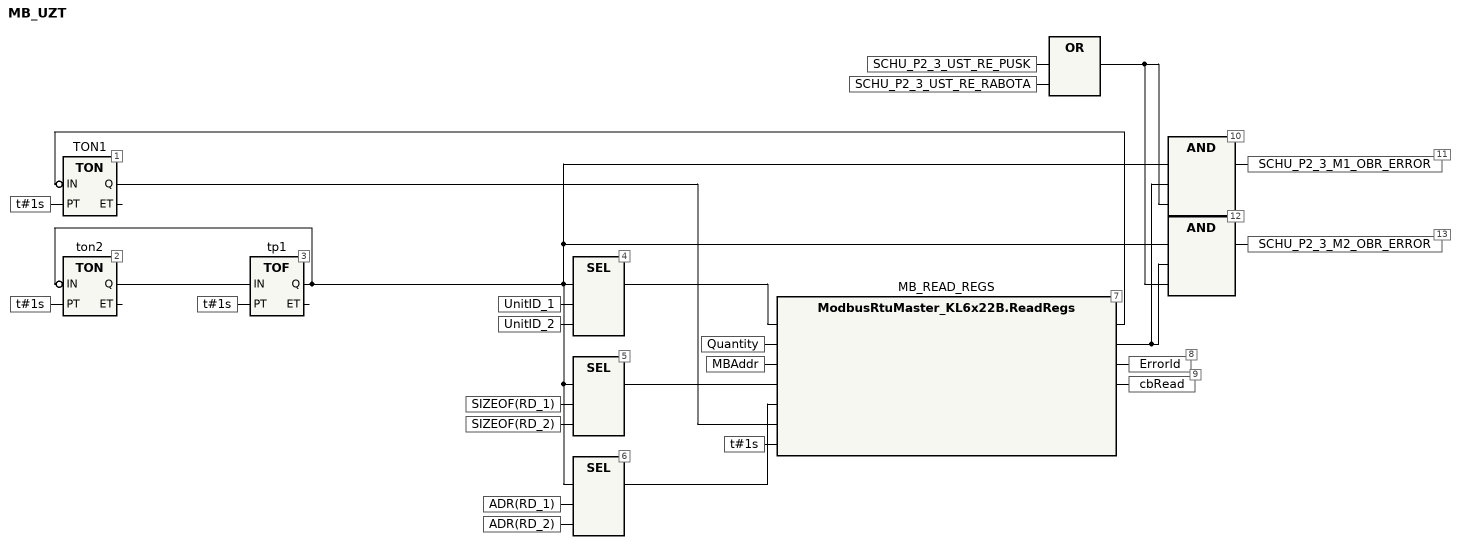
[picture p552: MB_UZT (CFC)]
_CFC_ (* Continuous Function Chart, elements in execution order *)
#0 OR(SCHU_P2_3_UST_RE_PUSK, SCHU_P2_3_UST_RE_RABOTA)
#1 TON1:TON(IN: NOT #7.out 1, PT: t#1s)
#2 ton2:TON(IN: NOT #3.Q, PT: t#1s)
#3 tp1:TOF(IN: #2.Q, PT: t#1s)
#4 SEL(#3.Q, UnitID_1, UnitID_2)
#5 SEL(#3.Q, SIZEOF(RD_1), SIZEOF(RD_2))
#6 SEL(#3.Q, ADR(RD_1), ADR(RD_2))
#7 MB_READ_REGS:ModbusRtuMaster_KL6x22B.ReadRegs(#4, Quantity, MBAddr, #5, #6, #1.Q, t#1s)
#8 Errorld <= #7.out 3
#9 cbRead <= #7.out 4
#10 AND(#3.Q, #7.out 2, #0)
#11 SCHU_P2_3_M1_OBR_ERROR <= #10
#12 AND(#3.Q, #7.out 2, #0)
#13 SCHU_P2_3_M2_OBR_ERROR <= #12
_END_CFC_
END_PROGRAM

(* POU IM/YA1_Upr_1, CFC *)
PROGRAM YA1_Upr_1
VAR
	RS_YA1_Open: RS;
	RT_Pusk: R_TRIG;
	RT_OSTANOV: R_TRIG;
	fb_HVACPA: FB_HVAC2PointActuator;

	stokeTime: TIME;
	enableLimitSwitch: BOOL := TRUE;
	FT_PCH_OTKL: R_TRIG;
	TON_PCH_OTKL: TON;
	ZADERJ_SHOD_YA1: TON;
	TON_YA1_Z_ZAM_TE2: TON;
	TON_OTK_MV: TON;
END_VAR
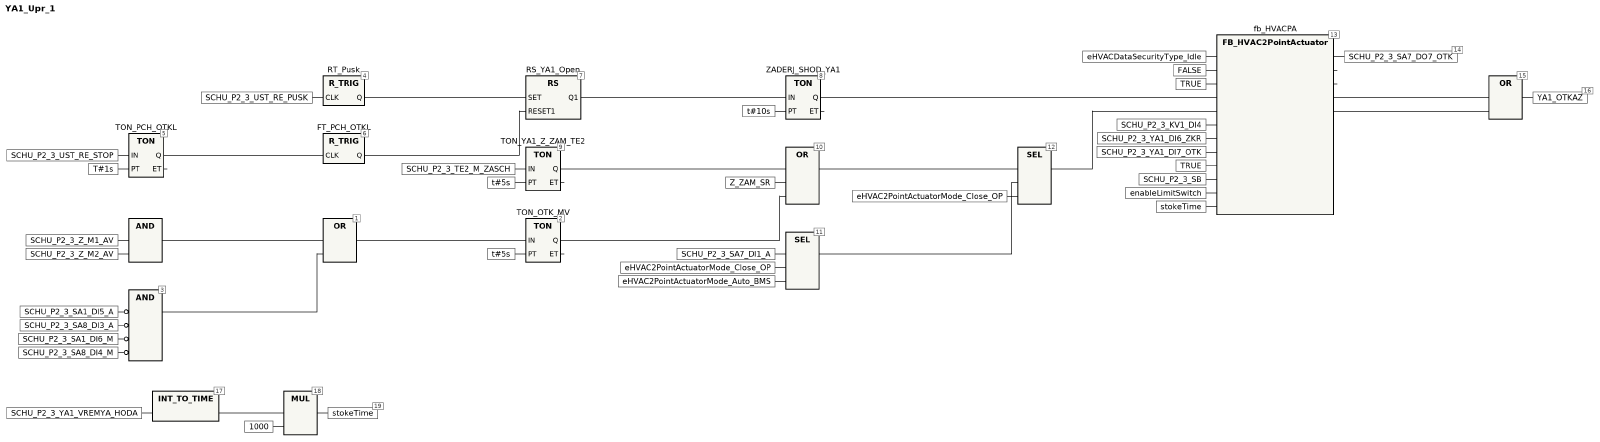
